# EPICS autosave request: ADApp/Db/NDDriverStdArrays_settings.req
file "ADBase_settings.req", P=$(P), R=$(R)
$(P)$(R)ArrayMode
$(P)$(R)CallbackMode
